Universal Robots PolyScope program: Servoj_rtde_example.urp

Program Servoj_rtde_example (installation=3M_neum directory=/programs/usbdisk/CODE/rtde_servoj createdIn=3.2.19275.0 lastSavedIn=5.8.2.10297 robotSerialNumber=20195500516)
Calibrated DH parameters: a=[0.000086, -0.265179, -0.334799, -0.000075, 0.000093, 0]; d=[0.162635, -1081.758718, 1011.830709, 70.061676, 0.099733, 0.099582]; alpha=[1.570538, 0.000307, 0.002928, 1.570251, -1.570005, 0]; deltaTheta=[0, -0.897626, 6.632003, 0.54881, 0, -0.000001]
BeforeStart
  Script: write_output_boolean_register(0,  True )
  Wait Sleep waitTime=0.01
  mode := 0
  j := [0.,0,0,0,0,0]
Robot Program (runOnlyOnce=true)
  Script: write_output_boolean_register(0,  False )
  Script: mode = read_input_integer_register(0)
  Loop While (checkContinuously=false) expression=mode < 3
    Loop While (checkContinuously=false) expression=mode ≟ 1
      MoveJ speed 15 deg/s, acceleration 40 deg/s^2 (useActiveTCP=true) feature=Base
        Waypoint Waypoint (Variable): variable(name=j)
      Script: write_output_boolean_register(0, True )
      Script: mode = read_input_integer_register(0)
      Script: sync()
    Loop While (checkContinuously=false) expression=(mode ≟ 2)
      SuppressedNode
        Script: servoj(j, lookahead_time=0.05, gain=3000)
      Script: servoj(j)
      Script: mode = read_input_integer_register(0)
    Script: mode = read_input_integer_register(0)
    Script: sync()
Thread Thread_1 (runOnlyOnce=false)
  Loop Forever
    tmp := [0,0,0,0,0,0]
    Script: tmp[0] = read_input_float_register(0)
    Script: tmp[1] = read_input_float_register(1)
    Script: tmp[2] = read_input_float_register(2)
    Script: tmp[3] = read_input_float_register(3)
    Script: tmp[4] = read_input_float_register(4)
    Script: tmp[5] = read_input_float_register(5)
    j := tmp
    Script: sync()
